FUNCTION TryConvert_WORD_TO_SINT : BOOL
VAR_INPUT
	in : WORD;
	out : REFERENCE TO SINT;
END_VAR

IF in > DatatypeLimits.MAX_VALUE_OF_WORD_WHICH_CAN_BE_HELD_IN_A_SINT THEN
	RETURN;
END_IF

out := WORD_TO_SINT(in);
TryConvert_WORD_TO_SINT := TRUE;

END_FUNCTION

(* stored: Version 1.1.0.1, ProductVersion 3.1.4024.12
   POU TryConvert_WORD_TO_SINT: Id {bddbb298-04ff-461e-b256-a2be75144a90}, SpecialFunc None *)
